INTERFACE I_HardwarePool

METHOD registerPc : BOOL
VAR_INPUT
  sNewPc : POINTER TO FB_PC;
  //pAdsConfig  : POINTER TO FB_ADS_Config;
END_VAR
END_METHOD

METHOD registerPh : BOOL
VAR_INPUT
    pNewPh       : POINTER TO FB_PH;
    //pAdsConfig   : POINTER TO FB_ADS_Config;
    //pConnectedCb : POINTER TO CalmarCompPrint.FB_PC;
    //iChannel     : INT;
END_VAR
END_METHOD

END_INTERFACE

(* stored: Version 1.1.0.1, ProductVersion 3.1.4024.11
   Itf I_HardwarePool: Id {b4c5cd3d-5e91-4396-bf52-168caeb885c5}
   Method registerPc: Id {2a3c4c0e-2ebc-446e-bd59-919efea24de5}
   Method registerPh: Id {8a0a5ac0-51d0-4726-a9f5-18888bbb4870} *)
